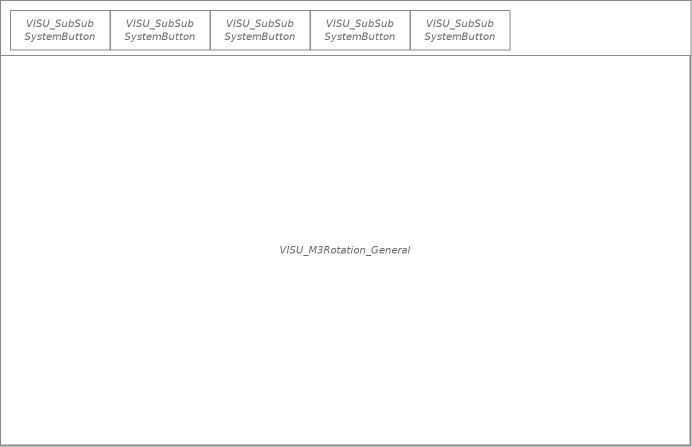
VISUALIZATION VISU_M3Rotation  // 692x447
VAR_IN_OUT
	ref : M3Rotation;
    widget : M3RotationWidget;
    m3Ref : M3;
    m3Widget : M3Widget;
END_VAR
    Frame (0,55 690x390), frame switch variable: widget.activeTab
        shows VISU_M3Rotation_General(ref := ref, widget := widget, m3Ref := m3Ref, m3Widget := m3Widget)
        shows VISU_AngularAxis(axis := ref.parts.positioningAxis, widget := widget.positioningAxis)
        shows VISU_FaulhaberDrive(drive := ref.parts.positioningDrive, widget := widget.positioningDrive)
        shows VISU_AngularAxis(axis := ref.parts.antiBacklashAxis, widget := widget.antiBacklashAxis)
        shows VISU_FaulhaberDrive(drive := ref.parts.antiBacklashDrive, widget := widget.antiBacklashDrive)
        p3374720746: ref.parts.positioningDrive
        p2332238231: ref.parts.antiBacklashDrive
    Frame (10,10 100x40)
        shows VISU_SubSubSystemButton(widget := widget.button_general)
        OnMouseClick: FrameSelectionChange Selection=SelectedFrame=1ceb887c-2a9b-46e4-a445-332726b96d42, GlobSel=AssignType=Directly, SelType=Locally
        OnMouseClick: execute { widget.activeTab := 0; }
    Frame (110,10 100x40)
        shows VISU_SubSubSystemButton(widget := widget.button_posAxis)
        OnMouseClick: FrameSelectionChange Selection=SelectedFrame=1ceb887c-2a9b-46e4-a445-332726b96d42, Selection=1, GlobSel=AssignType=Directly, SelType=Locally
        OnMouseClick: execute { widget.activeTab := 1; }
    Frame (210,10 100x40)
        shows VISU_SubSubSystemButton(widget := widget.button_posDrive)
        OnMouseClick: FrameSelectionChange Selection=SelectedFrame=1ceb887c-2a9b-46e4-a445-332726b96d42, Selection=2, GlobSel=AssignType=Directly, SelType=Locally
        OnMouseClick: execute { widget.activeTab := 2; }
    Frame (310,10 100x40)
        shows VISU_SubSubSystemButton(widget := widget.button_ablAxis)
        OnMouseClick: FrameSelectionChange Selection=SelectedFrame=1ceb887c-2a9b-46e4-a445-332726b96d42, Selection=3, GlobSel=AssignType=Directly, SelType=Locally
        OnMouseClick: execute { widget.activeTab := 3; }
    Frame (410,10 100x40)
        shows VISU_SubSubSystemButton(widget := widget.button_ablDrive)
        OnMouseClick: FrameSelectionChange Selection=SelectedFrame=1ceb887c-2a9b-46e4-a445-332726b96d42, Selection=4, GlobSel=AssignType=Directly, SelType=Locally
        OnMouseClick: execute { widget.activeTab := 4; }
END_VISUALIZATION

(* stored: Version 1.1.0.1, ProductVersion 3.1.4019.2
   Visu VISU_M3Rotation: Id {f87d7a58-379c-4af5-821e-afc5796615bf} *)
